// TwinCAT 3 PLC project Untitled1
// ProgramVersion: 3.1.4024.0
// libraries:
//   Tc2_Standard, * (Beckhoff Automation GmbH)
//   Tc2_System, * (Beckhoff Automation GmbH)
//   Tc3_Module, * (Beckhoff Automation GmbH)
// project tree:
//   / PlcTask.TcTTO
//   POUs/ FB_Camera.TcPOU, FB_ScannerImplementation.TcPOU, FB_ST45s.TcPOU, MAIN.TcPOU
// real-time tasks:
//   TASK PlcTask: cycle T#10ms, priority 20, ADS port 350

CONFIGURATION Untitled1
    RESOURCE PLC ON TwinCAT3
        TASK PlcTask(INTERVAL := T#10ms, PRIORITY := 20);
        PROGRAM MAIN WITH PlcTask : MAIN;
    END_RESOURCE
END_CONFIGURATION

// ---- POUs/MAIN.TcPOU
PROGRAM MAIN
VAR
	_Ivana : BOOL;
END_VAR

END_PROGRAM

// ---- POUs/FB_Camera.TcPOU
FUNCTION_BLOCK FB_Camera
VAR
	_IV3 : BOOL;
END_VAR

METHOD PROTECTED _scanner
VAR_INPUT
	_scanner : BOOL;
	_Keyence : BOOL;
	_Ivana	: BOOL;
END_VAR
END_METHOD

END_FUNCTION_BLOCK

// ---- POUs/FB_ScannerImplementation.TcPOU
FUNCTION_BLOCK FB_ScannerImplementation
VAR
	_Keyence : BOOL;
	_scannerCognex : BOOL;
END_VAR

_Keyence:= TRUE;

END_FUNCTION_BLOCK

// ---- POUs/FB_ST45s.TcPOU
FUNCTION_BLOCK FB_ST45s
VAR
	_camera : BOOL;
	_sensor	: BOOL;
END_VAR

END_FUNCTION_BLOCK
